# EPICS autosave request: quadEMApp/Db/quadEM_IOC_settings.req
file "quadEM_settings.req",            P=$(P), R=$(R)
file "quadEM_Plugin_settings.req",     P=$(P), R=$(R)
file "commonPlugin_settings.req",      P=$(P)
file "NDStdArrays_settings.req",       P=$(P), R=$(R)image1:
